(* PLC project ethernet_project.project, CODESYS CODESYS V3.5 SP8 Patch 2 *)
(* stored: creationDateTime 2016-04-24T20:19:19.2568173, modificationDateTime 2016-04-24T20:16:51.2703529 *)

PROGRAM fuzzy_exp_arab
  VAR
    e : INT := 0;
    a : INT := 10;
    b : INT := 20;
    c : INT := 30;
    d : INT := 40;
    f : INT := 0;
    g : INT := 50;
    h : INT := 100;
    xa : INT := 0;
    xb : INT := 30;
    xc : INT := 60;
  END_VAR
  VAR_INPUT
    temp : INT := 10;
    moist : INT := 10;
  END_VAR
  VAR
    cold : INT := 0;
    cool : INT := 0;
    normal : INT := 0;
    warm : INT := 0;
    hot : INT := 0;
    dry : INT := 0;
    most : INT := 0;
    wet : INT := 0;
    r1 : INT;
    r2 : INT;
    r3 : INT;
    r4 : INT;
    r5 : INT;
    k1 : INT;
    k2 : INT;
    k3 : INT;
    kk4 : INT;
    r6 : INT;
    r9 : INT;
    r7 : INT;
    r10 : INT;
    r8 : INT;
    r11 : INT;
    k8 : INT;
    k9 : INT;
    k10 : INT;
    k11 : INT;
    kk12 : INT;
    r12 : INT;
    r13 : INT;
    r15 : INT;
    r14 : INT;
    k5 : INT;
    k6 : INT;
    kk7 : INT;
    time_t : INT;
    moistvaltas : INT := 1;
    modulus : INT;
    time_nagyobb_0anal : INT := 0;
    tempvaltas : INT := 10;
  END_VAR

                    //t:=input('temp'); --eredeti
//t:=STRING_TO_INT('temp');
//moist:=input('رطوبة '); --eredeti
//moist:= STRING_TO_INT('رطوبة ');

// fuzzifation مرحلة تمثيل
IF temp<e THEN
    cold:=1;
ELSIF temp>=e AND temp<a THEN
	cold:=(a-temp)/(a-e);
    cool:=(temp-e)/(a-e);
ELSIF temp>=a AND temp<b THEN
    cool:=(b-temp)/(b-a);
    normal:=(temp-a)/(b-a);
ELSIF temp>=b AND temp<c THEN
	normal:=(c-temp)/(c-b);
	warm:=(temp-b)/(c-b);
ELSIF temp>=c AND temp<d THEN
	warm:=(d-temp)/(d-c);
    hot:=(temp-c)/(d-c);
else
    hot:=1;
END_IF;
IF moist<f THEN
	dry:=1;
ELSIF moist>=f AND moist<g THEN
    dry:=(g-moist)/(g-f);
	most:=(moist-f)/(g-f);
ELSIF moist>=g AND moist<h THEN
	most:=(h-moist)/(h-g);
	wet:=(moist-g)/(h-g);
else
    wet:=1;
END_IF;
//max.min and rulebaseمرحلة 
//for short
r1:=MIN (most,cold);
r2:=MIN (wet,cold);
r3:=MIN (wet,cool);
r4:=MIN (wet,normal);
r5:=MIN (wet,warm);
k1:=MAX(r1,r2);
k2:=MAX(k1,r3);
k3:=MAX(r4,r5);
kk4:=MAX(k2,k3);
//for midium
r6:=MIN (dry,cold);
r9:=MIN (most,normal);
r7:=MIN (most,cool);
r10:=MIN (most,hot);
r8:=MIN (most,warm);
r11:=MIN (wet,hot);
k8:=MAX(r6,r9);
k9:=MAX(r7,r10);
k10:=MAX(r8,r11);
k11:=MAX(k8,k9);
kk12:=MAX(k11,k10);
//for long
r12:=MIN (dry,hot);
r13:=MIN (dry,warm);
r15:=MIN (dry,cool);
r14:=MIN (dry,normal);
k5:=MAX(r12,r14);
k6:=MAX(r13,r15);
kk7:=MAX(k5,k6);
//defuzzification
IF (kk4+kk12+kk7) > 0 THEN
	time_t := (kk4*xa+kk12*xb+kk7*xc) / (kk4+kk12+kk7);
ELSE 
	time_t := -22;
END_IF;

IF temp >= 100 OR temp <= 0 THEN
	tempvaltas := tempvaltas * -1;	
END_IF;

//IF moist <= 0 OR moist >= 40 THEN
	//moistvaltas := moistvaltas * -1;
//END_IF
//moist := moist + moistvaltas;

IF time_t > 0 THEN
	time_nagyobb_0anal := time_nagyobb_0anal + 1;
END_IF
temp := temp + tempvaltas;

                  
END_PROGRAM

(* @NESTEDCOMMENTS := 'Yes' @PATH := '' @SYMFILEFLAGS := '2048' *)
FUNCTION_BLOCK masodik_fuzzy
  VAR_INPUT
    PV : REAL;
    SP : REAL;
    MV_LN : REAL;
    MV_MN : REAL;
    MV_SN : REAL;
    MV_SP : REAL;
    MV_MP : REAL;
    MV_LP : REAL;
    LN_Error_Rate : REAL;
    MN_Error_Rate : REAL;
    MP_Error_Rate : REAL;
    LP_Error_Rate : REAL;
    Update_Time : WORD;
    Manual : BOOL;
    CV_Manual : REAL;
    CV_Min : REAL;
    CV_Max : REAL;
    Enable : BOOL;
  END_VAR
  VAR_OUTPUT
    FL_CV : REAL;
  END_VAR
  VAR
    Loop_Update_ONS : R_TRIG;
    Loop_Update_Trigger : BOOL;
    TMR_Loop_Update : TON;
    Loop_Update_Time : WORD;
    Loop_Update_mSec : TIME;
    Process_Error : REAL;
    NL_Error : BOOL;
    NM_Error : BOOL;
    NS_Error : BOOL;
    PS_Error : BOOL;
    PM_Error : BOOL;
    PL_Error : BOOL;
    Process_Error_Rate : REAL;
    Error_Rate_PV1 : REAL;
    Error_Rate_PV2 : REAL;
    NL_Error_Rate_Ind : BOOL;
    NM_Error_Rate_Ind : BOOL;
    NS_Error_Rate_Ind : BOOL;
    PS_Error_Rate_Ind : BOOL;
    PM_Error_Rate_Ind : BOOL;
    PL_Error_Rate_Ind : BOOL;
    Output_CV : REAL;
  END_VAR

                    (* @END_DECLARATION := '0' *)
(****************************************************************************************************************************
	POU Title:  	Fuzzy_Logic(PRG)
   
 	Designer:	K. Presssley
	Date:		01/09/09
		
	Function:	The function of this program is to implement a fuzzy logic control algorithm for process control..  
****************************************************************************************************************************)
(***** Loop Update Logic *****)
(*  Get the Loop Update Time, ensure that lower limit of 1 is not exceeded and convert it into a time variable  *)
	IF Update_Time < 1 THEN
		Loop_Update_Time := 1;
	ELSE
		Loop_Update_Time := Update_Time;
	END_IF;

	Loop_Update_mSec := WORD_TO_TIME(Loop_Update_Time);

	IF NOT TMR_Loop_Update.Q THEN
		Loop_Update_Trigger := TRUE;
	ELSE
		Loop_Update_Trigger := FALSE;
	END_IF;

	TMR_Loop_Update( IN := Loop_Update_Trigger, PT:= Loop_Update_mSec );
 	  Loop_Update_ONS( CLK := TMR_Loop_Update.Q);



(***** Calculate the Process Error and Process Error Rate *****)
	IF Loop_Update_ONS.Q THEN
	  (* Process Error Calculation *)
		Process_Error := SP - PV;

	  (* Process Error Rate Calculation *)
	 	Error_Rate_PV1 := Error_Rate_PV2;
		  Error_Rate_PV2 := PV;
		   Process_Error_Rate := (Error_Rate_PV2 - Error_Rate_PV1) / (Loop_Update_Time);
	END_IF;


(***** Membership Zone Logic *****)
(* Error Zone Identification Logic - This logic will indentify which Error Zone the Process Value is currently in *)
	(* Negative Large Membership Zone *)
		IF Process_Error <= MV_LN THEN
			NL_Error := TRUE;
		ELSE
			NL_Error := FALSE;
		END_IF;

	(* Negative Medium Membership Zone *)
		IF Process_Error > MV_LN AND Process_Error <= MV_MN THEN
			NM_Error := TRUE;
		ELSE
			NM_Error := FALSE;
		END_IF;

	(* Negative Small Membership Zone *)
		IF Process_Error > MV_MN AND Process_Error <= MV_SN THEN
			NS_Error := TRUE;
		ELSE
			NS_Error := FALSE;
		END_IF;

	(* Positive Small Membership Zone *)
		IF Process_Error < MV_MP AND Process_Error >= MV_SP THEN
			PS_Error := TRUE;
		ELSE
			PS_Error := FALSE;
		END_IF;

	(* Positive Medium Membership Zone *)
		IF Process_Error < MV_LP AND Process_Error >= MV_MP THEN
			PM_Error := TRUE;
		ELSE
			PM_Error := FALSE;
		END_IF;

	(* Positive Large Membership Zone *)
		IF Process_Error >= MV_LP THEN
			PL_Error := TRUE;
		ELSE
			PL_Error := FALSE;
		END_IF;

(* Error Rate Zone Identification Logic - This logic will indentify which Error Rate Zone the Process Value is currently in *)
	(* Negative Large Error Rate Membership Zone - The Error Rate is Decreasing Quickly *)
		IF Process_Error_Rate <= LN_Error_Rate THEN
			NL_Error_Rate_Ind := TRUE;
		ELSE
			NL_Error_Rate_Ind := FALSE;
		END_IF;

	(* Negative Medium Error Rate Membership Zone - The Error Rate is Decreasing *)
		IF Process_Error_Rate > LN_Error_Rate AND Process_Error_Rate <= MN_Error_Rate THEN
			NM_Error_Rate_Ind := TRUE;
		ELSE
			NM_Error_Rate_Ind := FALSE;
		END_IF;

	(* Negative Small Error Rate Membership Zone  - The Error Rate is Decreasing slowly *)
		IF Process_Error_Rate > MN_Error_Rate AND Process_Error_Rate < 0.0 THEN
			NS_Error_Rate_Ind := TRUE;
		ELSE
			NS_Error_Rate_Ind := FALSE;
		END_IF;

	(* Positive Small Error Rate Membership Zone  - The Error Rate is Increasing slowly *)
		IF Process_Error_Rate < MP_Error_Rate AND Process_Error_Rate >= 0.0 THEN
			PS_Error_Rate_Ind := TRUE;
		ELSE
			PS_Error_Rate_Ind := FALSE;
		END_IF;

	(* Positive Meduim Error Rate Membership Zone  - The Error Rate is Increasing *)
		IF Process_Error_Rate < LP_Error_Rate AND Process_Error_Rate >= MP_Error_Rate THEN
			PM_Error_Rate_Ind := TRUE;
		ELSE
			PM_Error_Rate_Ind := FALSE;
		END_IF;

	(* Positive Large Error Rate Membership Zone  - The Error Rate is Increasing Quickly  *)
		IF Process_Error_Rate >= LP_Error_Rate THEN
			PL_Error_Rate_Ind := TRUE;
		ELSE
			PL_Error_Rate_Ind := FALSE;
		END_IF;


(***** Fuzzy Logic Rules *****)
(* This section of logic contains all of the Fuzzy Logic rules required to produce the control action *)
	(* PV is Far Above SP and Increasing Quickly *)
		IF Loop_Update_ONS.Q AND NL_Error AND PL_Error_Rate_Ind
		    AND Enable AND NOT Manual THEN
			Output_CV := Output_CV - 1000.0;
		END_IF;

	(* PV is Far Above SP and Increasing *)
		IF Loop_Update_ONS.Q AND NL_Error AND PM_Error_Rate_Ind
		    AND Enable AND NOT Manual THEN
			Output_CV := Output_CV - 300.0;
		END_IF;

	(* PV is Far Above SP and Increasing slowly *)
		IF Loop_Update_ONS.Q AND NL_Error AND PS_Error_Rate_Ind
		    AND Enable AND NOT Manual THEN
			Output_CV := Output_CV - 250.0;
		END_IF;

	(* PV is Far Above SP and Decreasing slowly *)
		IF Loop_Update_ONS.Q AND NL_Error AND NS_Error_Rate_Ind
		    AND Enable AND NOT Manual THEN
			Output_CV := Output_CV - 300;
		END_IF;

	(* PV is Far Above SP and Decreasing *)
		IF Loop_Update_ONS.Q AND NL_Error AND NM_Error_Rate_Ind
		    AND Enable AND NOT Manual THEN
			Output_CV := Output_CV - 250.0;
		END_IF;

	(* PV is Far Above SP and Decreasing Quickly *)
		IF Loop_Update_ONS.Q AND NL_Error AND NL_Error_Rate_Ind
		    AND Enable AND NOT Manual THEN
			Output_CV := Output_CV - 100.0;
		END_IF;

	(* PV is Above SP and Increasing Quickly *)
		IF Loop_Update_ONS.Q AND NM_Error AND PL_Error_Rate_Ind
		    AND Enable AND NOT Manual THEN
			Output_CV := Output_CV - 250.0;
		END_IF;

	(* PV is Above SP and Increasing *)
		IF Loop_Update_ONS.Q AND NM_Error AND PM_Error_Rate_Ind
		    AND Enable AND NOT Manual THEN
			Output_CV := Output_CV - 100.0;
		END_IF;

	(* PV is Above SP and Increasing slowly *)
		IF Loop_Update_ONS.Q AND NM_Error AND PS_Error_Rate_Ind
		    AND Enable AND NOT Manual THEN
			Output_CV := Output_CV - 50.0;
		END_IF;

	(* PV is Above SP and Decreasing Slowly *)
		IF Loop_Update_ONS.Q AND NM_Error AND NS_Error_Rate_Ind
		    AND Enable AND NOT Manual THEN
			Output_CV := Output_CV - 250.0;
		END_IF;

	(* PV is Above SP and Decreasing *)
		IF Loop_Update_ONS.Q AND NM_Error AND NM_Error_Rate_Ind
		    AND Enable AND NOT Manual THEN
			Output_CV := Output_CV - 100.0;
		END_IF;

	(* PV is Above SP and Decreasing Quickly *)
		IF Loop_Update_ONS.Q AND NM_Error AND NL_Error_Rate_Ind
		    AND Enable AND NOT Manual THEN
			Output_CV := Output_CV - 50.0;
		END_IF;

	(* PV is Slightly Above SP and Increasing Quickly *)
		IF Loop_Update_ONS.Q AND NS_Error AND PL_Error_Rate_Ind
		    AND Enable AND NOT Manual THEN
			Output_CV := Output_CV - 20.0;
		END_IF;

	(* PV is Slightly Above SP and Increasing *)
		IF Loop_Update_ONS.Q AND NS_Error AND PM_Error_Rate_Ind
		    AND Enable AND NOT Manual THEN
			Output_CV := Output_CV - 10.0;
		END_IF;

	(* PV is Slightly Above SP and Increasing slowly*)
		IF Loop_Update_ONS.Q AND NS_Error AND PS_Error_Rate_Ind
		    AND Enable AND NOT Manual THEN
			Output_CV := Output_CV - 5.0;
		END_IF;

	(* PV is Slightly Above SP and Decreasing slowly*)
		IF Loop_Update_ONS.Q AND NS_Error AND NS_Error_Rate_Ind
		    AND Enable AND NOT Manual THEN
			Output_CV := Output_CV - 20.0;
		END_IF;

	(* PV is Slightly Above SP and Decreasing *)
		IF Loop_Update_ONS.Q AND NS_Error AND NM_Error_Rate_Ind
		    AND Enable AND NOT Manual THEN
			Output_CV := Output_CV - 10.0;
		END_IF;

	(* PV is Slightly Above SP and Decreasing Quickly*)
		IF Loop_Update_ONS.Q AND NS_Error AND NL_Error_Rate_Ind
		    AND Enable AND NOT Manual THEN
			Output_CV := Output_CV - 5.0;
		END_IF;

	(* PV is Slightly Below SP and Increasing Quickly *)
		IF Loop_Update_ONS.Q AND PS_Error AND PL_Error_Rate_Ind
		    AND Enable AND NOT Manual THEN
			Output_CV := Output_CV + 5.0;
		END_IF;

	(* PV is Slightly Below SP and Increasing *)
		IF Loop_Update_ONS.Q AND PS_Error AND PM_Error_Rate_Ind
		    AND Enable AND NOT Manual THEN
			Output_CV := Output_CV + 10.0;
		END_IF;

	(* PV is Slightly Below SP and Increasing Slowly *)
		IF Loop_Update_ONS.Q AND PS_Error AND PS_Error_Rate_Ind
		    AND Enable AND NOT Manual THEN
			Output_CV := Output_CV + 20.0;
		END_IF;

	(* PV is Slightly Below SP and Decreasing Slowly *)
		IF Loop_Update_ONS.Q AND PS_Error AND NS_Error_Rate_Ind
		    AND Enable AND NOT Manual THEN
			Output_CV := Output_CV + 20.0;
		END_IF;

	(* PV is Slightly Below SP and Decreasing *)
		IF Loop_Update_ONS.Q AND PS_Error AND NM_Error_Rate_Ind
		    AND Enable AND NOT Manual THEN
			Output_CV := Output_CV + 10.0;
		END_IF;

	(* PV is Slightly Below SP and Decreasing Quickly *)
		IF Loop_Update_ONS.Q AND PS_Error AND NL_Error_Rate_Ind
		    AND Enable AND NOT Manual THEN
			Output_CV := Output_CV + 5.0;
		END_IF;

	(* PV is Below SP and Increasing Quickly *)
		IF Loop_Update_ONS.Q AND PM_Error AND PL_Error_Rate_Ind
		    AND Enable AND NOT Manual THEN
			Output_CV := Output_CV + 50.0;
		END_IF;

	(* PV is Below SP and Increasing *)
		IF Loop_Update_ONS.Q AND PM_Error AND PM_Error_Rate_Ind
		    AND Enable AND NOT Manual THEN
			Output_CV := Output_CV + 20.0;
		END_IF;

	(* PV is Below SP and Increasing Slowly *)
		IF Loop_Update_ONS.Q AND PM_Error AND PS_Error_Rate_Ind
		    AND Enable AND NOT Manual THEN
			Output_CV := Output_CV + 10.0;
		END_IF;

	(* PV is Below SP and Decreasing Slowly *)
		IF Loop_Update_ONS.Q AND PM_Error AND NS_Error_Rate_Ind
		    AND Enable AND NOT Manual THEN
			Output_CV := Output_CV + 50.0;
		END_IF;

	(* PV is Below SP and Decreasing *)
		IF Loop_Update_ONS.Q AND PM_Error AND NM_Error_Rate_Ind
		    AND Enable AND NOT Manual THEN
			Output_CV := Output_CV + 100.0;
		END_IF;

	(* PV is Below SP and Decreasing Quickly *)
		IF Loop_Update_ONS.Q AND PM_Error AND NL_Error_Rate_Ind
		    AND Enable AND NOT Manual THEN
			Output_CV := Output_CV + 250.0;
		END_IF;

	(* PV is Far Below SP and Increasing Quickly *)
		IF Loop_Update_ONS.Q AND PL_Error AND PL_Error_Rate_Ind
		    AND Enable AND NOT Manual THEN
			Output_CV := Output_CV + 100.0;
		END_IF;

	(* PV is Far Below SP and Increasing *)
		IF Loop_Update_ONS.Q AND PL_Error AND PM_Error_Rate_Ind
		    AND Enable AND NOT Manual THEN
			Output_CV := Output_CV + 250.0;
		END_IF;

	(* PV is Far Below SP and Increasing Slowly *)
		IF Loop_Update_ONS.Q AND PL_Error AND PS_Error_Rate_Ind
		    AND Enable AND NOT Manual THEN
			Output_CV := Output_CV + 300.0;
		END_IF;

	(* PV is Far Below SP and Decreasing Slowly *)
		IF Loop_Update_ONS.Q AND PL_Error AND NS_Error_Rate_Ind
		    AND Enable AND NOT Manual THEN
			Output_CV := Output_CV + 100.0;
		END_IF;

	(* PV is Far Below SP and Decreasing *)
		IF Loop_Update_ONS.Q AND PL_Error AND NM_Error_Rate_Ind
		    AND Enable AND NOT Manual THEN
			Output_CV := Output_CV + 250.0;
		END_IF;

	(* PV is Far Below SP and Decreasing Quickly *)
		IF Loop_Update_ONS.Q AND PL_Error AND NL_Error_Rate_Ind
		    AND Enable AND NOT Manual THEN
			Output_CV := Output_CV + 300.0;
		END_IF;

	(* Write Output_CV to the controller output variable, CV *)
		IF Enable AND NOT Manual THEN
			FL_CV := Output_CV;
		END_IF;


(***** Fuzzy Logic Controller Maximum and Minimum Limits Logic *****)
(* Minimum Limits Logic *)
	IF Output_CV < CV_Min THEN
		Output_CV := CV_Min;
	END_IF;

(* Maximum Limits Logic *)
	IF Output_CV > CV_Max THEN
		Output_CV := CV_Max;
	END_IF;

(***** Manual Fuzzy Logic Controller Operation *****)
(* This section of logic controls the manual operation of the fuzzy logic controller.  If the controller
    is enabled and the manual control is set to True, then the output of the controller, CV, will be
    equal to CV_Manual. *)
	IF Enable AND Manual AND (CV_Manual > 0.0 AND CV_Manual <= 32767) THEN
		FL_CV := CV_Manual;
	END_IF;

	IF Enable AND Manual AND (CV_Manual < 0.0) THEN
		FL_CV := 0.0;
	END_IF;

	IF Enable AND Manual AND (CV_Manual >32767.0) THEN
		FL_CV := 32767.0;
	END_IF;

(* Fuzzy Logic Controller Enable Logic *)
	IF NOT Enable THEN
		Output_CV := 0.0;
		  FL_CV := 0.0;
	END_IF;

                  
END_FUNCTION_BLOCK

PROGRAM fuzzy_st
  VAR
    in1 : BOOL;
  END_VAR

                    
                  
END_PROGRAM

CONFIGURATION With_ethernet
  RESOURCE Application ON PLC
    TASK ExampleTask(INTERVAL := T#20ms, PRIORITY := 1);
    PROGRAM fuzzy_st WITH ExampleTask : fuzzy_st;
  END_RESOURCE
END_CONFIGURATION

CONFIGURATION EthernetModul
END_CONFIGURATION
